// SIMATIC S7-200 project (STEP 7-Micro/WIN), CPU 224XP REL 02.01

SYMBOL_TABLE USER1
di_0_0           I0.0
di_0_1           I0.1
di_0_2           I0.2     // lazer_ON
di_0_3           I0.3
di_0_4           I0.4
di_0_5           I0.5
di_0_6           I0.6
di_0_7           I0.7
di_1_0           I1.0
di_1_1           I1.1
di_1_2           I1.2
di_1_3           I1.3
di_1_4           I1.4
di_1_5           I1.5
m0.0             M0.0
m0.1             M0.1
m0.2             M0.2
m0.3             M0.3
m0.4             M0.4
m0.5             M0.5
m0.6             M0.6
m0.7             M0.7
m1.0             M1.0
m1.1             M1.1
m1.2             M1.2
m1.3             M1.3
m1.4             M1.4
m1.5             M1.5
m1.6             M1.6
m1.7             M1.7
MB_DONE          M3.0
Port0_free_MB    M3.1
mb_start_delay   M3.2
reset_doze_nd1_all M4.0
reset_doze_nd2_all M4.1
reset_doze_all   M4.2
q_0_0            Q0.0
q_0_1            Q0.1
q_0_2            Q0.2
q_0_3            Q0.3
q_0_4            Q0.4
q_0_5            Q0.5
q_0_6            Q0.6
q_0_7            Q0.7
q_1_0            Q1.0
q_1_1            Q1.1
q_2_0            Q2.0
q_2_1            Q2.1
q_2_2            Q2.2
q_2_3            Q2.3
q_2_4            Q2.4
q_2_5            Q2.5
q_2_6            Q2.6
q_2_7            Q2.7
q_3_0            Q3.0
q_3_1            Q3.1
q_3_2            Q3.2
q_3_3            Q3.3
q_3_4            Q3.4
q_3_5            Q3.5
q_3_6            Q3.6
q_3_7            Q3.7
q_4_0            Q4.0
q_4_1            Q4.1
q_4_2            Q4.2
q_4_3            Q4.3
q_4_4            Q4.4
q_4_5            Q4.5
q_4_6            Q4.6
q_4_7            Q4.7
err_dh2          V50.3
err_LT1_min_dop  V50.4
err_LT1_max_dop  V50.5
err_memory       V50.6
err_one_param    V50.7
err_ai_FT1       V51.0
err_ai_FT2       V51.1
err_ai_LT1       V51.2
err_ai_PT1       V51.3
err_PT1_max_dop  V51.4
err_sa2_stop     V51.5
err_dh1_aft      V51.6
err_dh2_aft      V51.7
warn_LT1_min_work V54.0
warn_LT1_max_work V54.1
warn_PT1_min_work V54.2
warn_PT1_max_work V54.3
warn_reserv_nd1_start V54.4
warn_reserv_nd2_start V54.5
warn_port0_mb    V54.6
warn_port0_mb_init V54.7
MB_ERR_CODE_DONE VB12
err_one_param_item VB13
MB_ERR_CODE_INIT VB14
port0_mb_addr    VB15
port0_mb_parity  VB16
par27            VB300    // port0_mb_parity
par28            VB301    // port0_mb_addr
par29            VB302    // again_dh
par30            VB303
par31            VB304
par32            VB305
par33            VB306
I_16MA           VD66
port0_mb_baudrate VD154
par34            VD320    // port0_mb_baudrate
par35            VD324
par36            VD328
sum1             VD360
sum2             VD364
rez1             VD368
rez2             VD372
doze_nd1_from_start VD376
doze_nd1_all     VD380
doze_nd2_from_start VD384
doze_nd2_all     VD388
tmpp             VD392
ai_FT1           VW0
ai_FT2           VW2
ai_LT1           VW4
ai_PT1           VW6
g_errors_0       VW50
g_errors_1       VW52
g_warnings_0     VW54
g_warnings_1     VW56
MB_HR            VW58
I_3MA            VW60
I_4MA            VW62
mb_start_delay_value VW64
LT1_zero         VW70
LT1_range        VW72
LT1_min_work     VW74
LT1_max_work     VW76
LT1_min_dop      VW78
LT1_max_dop      VW80
PT1_zero         VW82
PT1_range        VW84
PT1_min_work     VW86
PT1_max_work     VW88
PT1_max_dop      VW90
FT1_range        VW92
FT2_range        VW94
time_out_dh      VW96
time_out_dh_s    VW98
reserve_nd_start_tout_s VW100
reserve_nd_start_tout VW102
mask_errors_0    VW106
mask_errors_1    VW108
mask_warnings_0  VW110
mask_warnings_1  VW112
nsh_timer_counter_sec VW114
nsh_work_time    VW116
nsh_cycle_time   VW118
again_dh         VW120
par01            VW200    // FT1_RANGE
par02            VW202    // FT2_RANGE
par03            VW204    // PT1_RANGE
par04            VW206    // LT1_RANGE
par05            VW208    // PT1_zero
par06            VW210    // LT1_zero
par07            VW212    // LT1_min_work
par08            VW214    // LT1_max_work
par09            VW216    // LT1_min_dop
par10            VW218    // LT1_max_dop
par11            VW220    // PT1_min_work
par12            VW222    // PT1_max_work
par13            VW224    // PT1_max_dop
par14            VW226    // nsh_work_time:VW66
par15            VW228    // nsh_cycle_time:VW68
par16            VW230    // reserve_nd_start_tout_s:VW100
par17            VW232    // time_out_dh_s:VW98
par18            VW234    // again_dh
par19            VW236
par20            VW238
par21            VW240
par22            VW242
par23            VW244
par24            VW246
par25            VW248
par26            VW250
flow             VW252
tmp              VW350
count            VW352
adder            VW354
total1           VW356
total2           VW358
END_SYMBOL_TABLE

SYMBOL_TABLE MB_HOLD
H_40001          VW500    // ai_FT1
H_40002          VW502    // ai_FT2
H_40003          VW504    // ai_LT1
H_40004          VW506    // ai_PT1
H_40005          VW508
H_40006          VW510
H_40007          VW512
H_40008          VW514
H_40009          VW516
H_40010          VW518
H_40011          VW520
H_40012          VW522
H_40013          VW524
H_40014          VW526
H_40015          VW528
H_40016          VW530
H_40017_0        V532.0   // лазер
H_40017_1        V532.1   // свет нло
H_40017_2        V532.2
H_40017_3        V532.3
H_40017_4        V532.4
H_40017_5        V532.5
H_40017_6        V532.6
H_40017_7        V532.7
H_40017_8        V533.0   // свет
H_40017_9        V533.1   // q0.1
H_40017_10       V533.2   // q0.2
H_40017_11       V533.3   // relay 16a
H_40017_12       V533.4   // q0.4
H_40017_13       V533.5   // светофор хранилище
H_40017_14       V533.6   // +12 под нло резерв
H_40017_15       V533.7   // дым п1
H_40018_0        V534.0   // red
H_40018_1        V534.1   // green
H_40018_2        V534.2   // blue
H_40018_3        V534.3   // вход в дезинфекцию
H_40018_4        V534.4   // жалюзи закрыть
H_40018_5        V534.5   // жалюзи открыть
H_40018_6        V534.6   // вход в квест
H_40018_7        V534.7   // уф лампы
H_40018_8        V535.0   // откр рубильник
H_40018_9        V535.1   // микроскоп
H_40018_10       V535.2   // нло движение
H_40018_11       V535.3   // помпа жизнеобесп
H_40018_12       V535.4   // red
H_40018_13       V535.5   // green
H_40018_14       V535.6   // blue
H_40018_15       V535.7   // вход в смотровую
H_40019_0        V536.0
H_40019_1        V536.1
H_40019_2        V536.2
H_40019_3        V536.3
H_40019_4        V536.4
H_40019_5        V536.5
H_40019_6        V536.6
H_40019_7        V536.7
H_40019_8        V537.0   // warn_LT1_min_work:V54.0
H_40019_9        V537.1   // warn_LT1_max_work:V54.1
H_40019_10       V537.2   // warn_PT1_min_work:V54.2
H_40019_11       V537.3   // warn_PT1_max_work:V54.3
H_40019_12       V537.4   // warn_reserv_nd1_start:V54.4
H_40019_13       V537.5   // warn_reserv_nd2_start:V54.5
H_40019_14       V537.6   // q_3_6:Q3.6 exit qvest
H_40019_15       V537.7   // warn_port0_mb_init:V54.7
H_40020_0        V538.0   // power_on:M1.0
H_40020_1        V538.1   // ND1:M1.1
H_40020_2        V538.2   // ND2:M1.2
H_40020_3        V538.3   // nsh_manual:M1.3
H_40020_4        V538.4   // nsh_mixer_mode:M1.7
H_40020_5        V538.5   // Both_nd_enable:M1.4
H_40020_6        V538.6   // nsh_mixer:M1.6
H_40020_7        V538.7   // nsh_current:M1.5
H_40020_8        V539.0   // modul 3 4.0
H_40020_9        V539.1   // modul 3 4.1
H_40020_10       V539.2   // modul 3.4.2
H_40020_11       V539.3   // modul 3.4.3
H_40020_12       V539.4   // modul 3.4.4
H_40020_13       V539.5   // modul 3.4.5
H_40020_14       V539.6   // modul 3.4.6
H_40020_15       V539.7   // modul 3.4.7
H_40021_0        V540.0
H_40021_1        V540.1
H_40022          VW542
H_40023_0        V544.0
H_40023_1        V544.1
H_40023_2        V544.2
H_40023_3        V544.3
H_40023_4        V544.4
H_40023_5        V544.5
H_40023_6        V544.6
H_40023_7        V544.7
H_40023_8        V545.0
H_40023_9        V545.1
H_40023_10       V545.2
H_40023_11       V545.3
H_40023_12       V545.4
H_40023_13       V545.5
H_40023_14       V545.6
H_40023_15       V545.7
H_40024_0        V546.0
H_40024_1        V546.1
H_40024_2        V546.2
H_40024_3        V546.3
H_40024_4        V546.4
H_40024_5        V546.5
H_40024_6        V546.6
H_40024_7        V546.7
H_40024_8        V547.0
H_40024_9        V547.1
H_40024_10       V547.2
H_40024_11       V547.3
H_40024_12       V547.4
H_40024_13       V547.5
H_40024_14       V547.6
H_40024_15       V547.7
Н_40025          VW548
Н_40026          VW550
Н_40027          VW552
H_40028          VW554
H_40029_0        V556.0
H_40029_1        V556.1
H_40029_2        V556.2
H_40029_3        V556.3
H_40029_4        V556.4
H_40029_5        V556.5
H_40029_6        V556.6
H_40029_7        V556.7
H_40029_8        V557.0
H_40029_9        V557.1
H_40029_10       V557.2
H_40029_11       V557.3
H_40029_12       V557.4
H_40029_13       V557.5
H_40029_14       V557.6
H_40029_15       V557.7
H_40030_0        V558.0   // --
H_40030_1        V558.1
H_40030_2        V558.2
H_40030_3        V558.3
H_40030_4        V558.4
H_40030_5        V558.5
H_40030_6        V558.6
H_40030_7        V558.7
H_40030_8        V559.0
H_40030_9        V559.1
H_40030_10       V559.2
H_40030_11       V559.3
H_40030_12       V559.4
H_40030_13       V559.5
H_40030_14       V559.6
H_40030_15       V559.7
END_SYMBOL_TABLE

SYMBOL_TABLE S7-200 Symbols
Always_On        SM0.0    // Always ON
First_Scan_On    SM0.1    // ON for the first scan cycle only
Clock_1s         SM0.5    // Clock pulse that is ON for 0.5 s, OFF for 0.5 s, for a duty cycle time of 1 s.
Pot0_Value       SMB28    // Set to value corresponding to analog adjustment 0.
END_SYMBOL_TABLE

ORGANIZATION_BLOCK MAIN:OB1
TITLE=PROGRAM COMMENTS
BEGIN
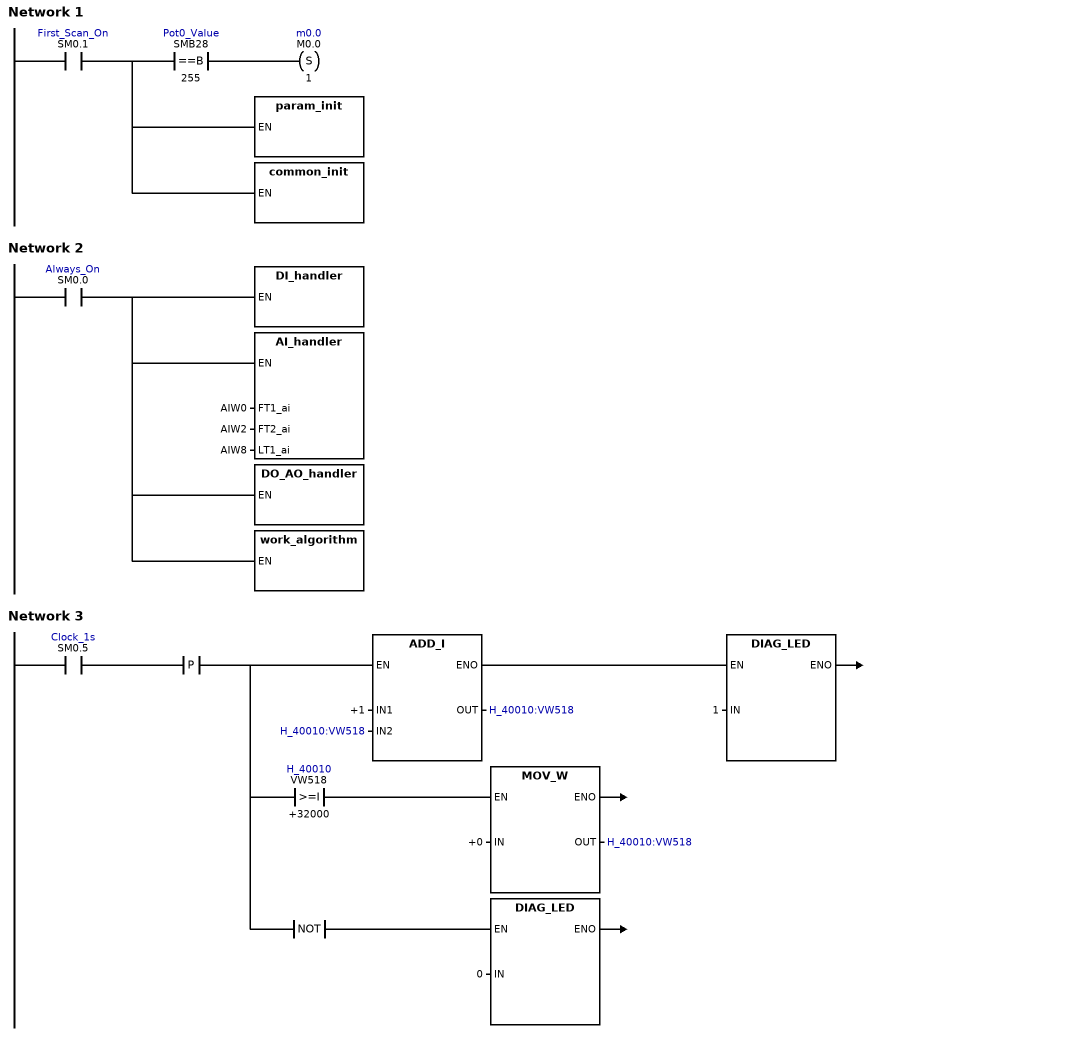
Network 1
LD     First_Scan_On:SM0.1
LPS
AB=    Pot0_Value:SMB28, 255
S      m0.0:M0.0, 1
LRD
CALL   param_init:SBR0
LPP
CALL   common_init:SBR1
Network 2
LD     Always_On:SM0.0
CALL   DI_handler:SBR2
CALL   AI_handler:SBR3, AIW0, AIW2, AIW8
CALL   DO_AO_handler:SBR6
CALL   work_algorithm:SBR4
Network 3
LD     Clock_1s:SM0.5
EU
LPS
+I     +1, H_40010:VW518
AENO
?32C   1
LRD
AW>=   H_40010:VW518, +32000
MOVW   +0, H_40010:VW518
LPP
NOT
?32C   0
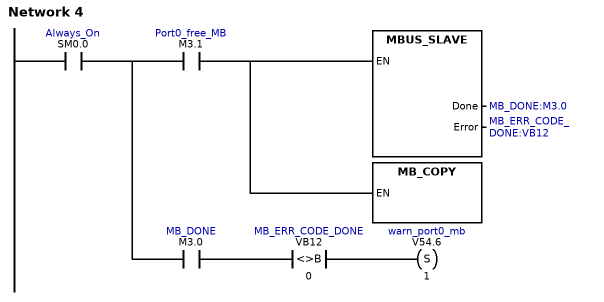
Network 4
LD     Always_On:SM0.0
LPS
A      Port0_free_MB:M3.1
CALL   MBUS_SLAVE:SBR13, MB_DONE:M3.0, MB_ERR_CODE_DONE:VB12
CALL   MB_COPY:SBR8
LPP
A      MB_DONE:M3.0
AB<>   MB_ERR_CODE_DONE:VB12, 0
S      warn_port0_mb:V54.6, 1
END_ORGANIZATION_BLOCK

SUBROUTINE_BLOCK param_init:SBR0
TITLE=
BEGIN
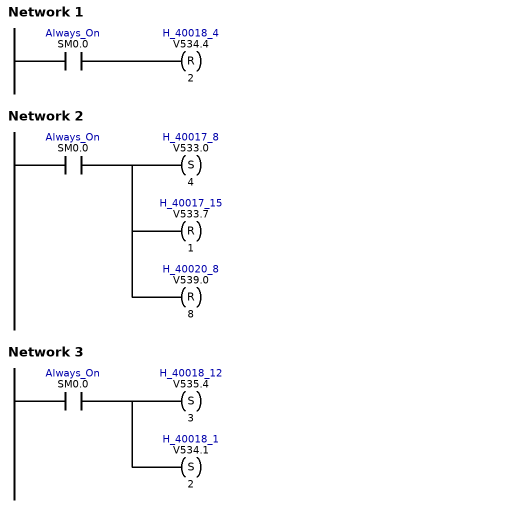
Network 1
LD     Always_On:SM0.0
R      H_40018_4:V534.4, 2
Network 2
LD     Always_On:SM0.0
S      H_40017_8:V533.0, 4
R      H_40017_15:V533.7, 1
R      H_40020_8:V539.0, 8
Network 3
LD     Always_On:SM0.0
S      H_40018_12:V535.4, 3
S      H_40018_1:V534.1, 2
END_SUBROUTINE_BLOCK

SUBROUTINE_BLOCK common_init:SBR1
TITLE=
BEGIN
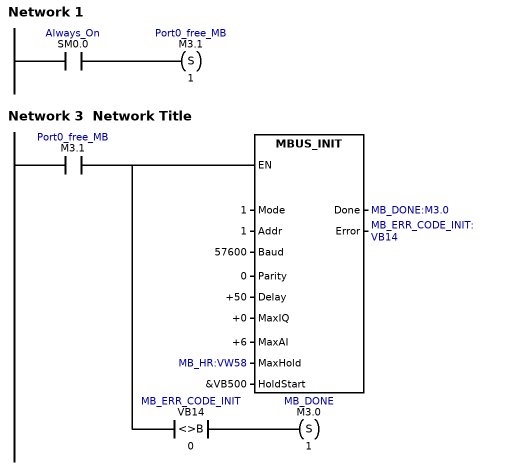
Network 1
LD     Always_On:SM0.0
S      Port0_free_MB:M3.1, 1
Network 3 // Network Title
LD     Port0_free_MB:M3.1
CALL   MBUS_INIT:SBR14, 1, 1, 57600, 0, +50, +0, +6, MB_HR:VW58, &VB500, MB_DONE:M3.0, MB_ERR_CODE_INIT:VB14
AB<>   MB_ERR_CODE_INIT:VB14, 0
S      MB_DONE:M3.0, 1
END_SUBROUTINE_BLOCK

SUBROUTINE_BLOCK AI_handler:SBR3
TITLE=SUBROUTINE COMMENTS
VAR_INPUT
FT1_ai:WORD;	// LW0 
FT2_ai:WORD;	// LW2 
LT1_ai:WORD;	// LW4 
END_VAR
BEGIN
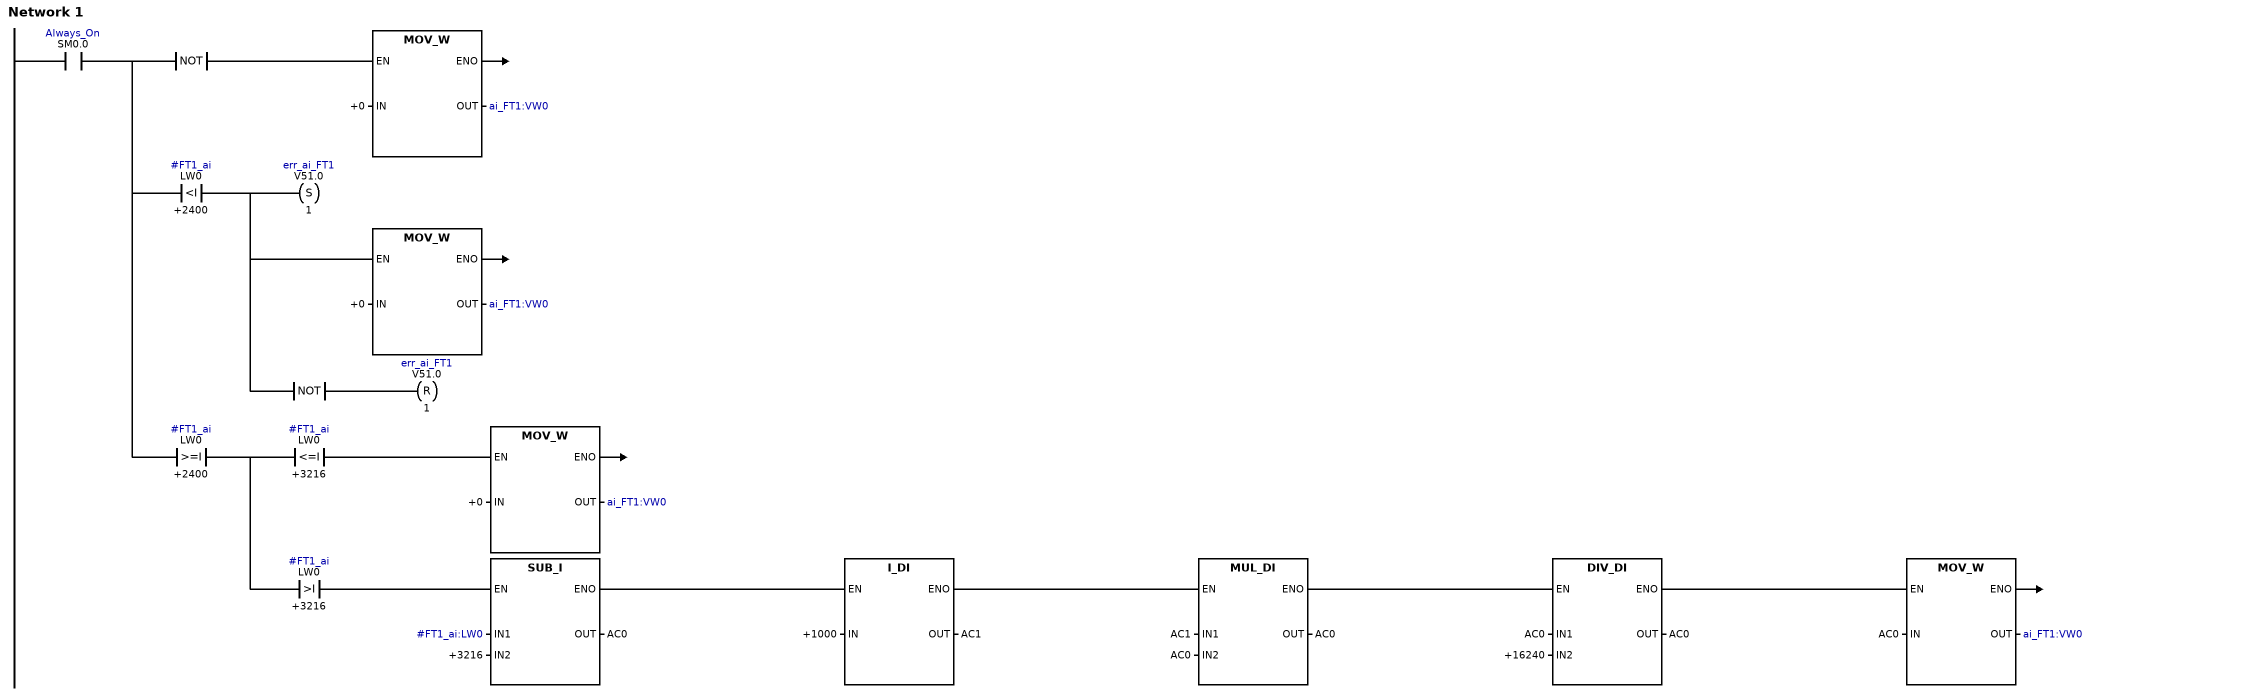
Network 1
LD     Always_On:SM0.0
LPS
NOT
MOVW   +0, ai_FT1:VW0
LRD
AW<    #FT1_ai:LW0, +2400
S      err_ai_FT1:V51.0, 1
MOVW   +0, ai_FT1:VW0
NOT
R      err_ai_FT1:V51.0, 1
LPP
AW>=   #FT1_ai:LW0, +2400
LPS
AW<=   #FT1_ai:LW0, +3216
MOVW   +0, ai_FT1:VW0
LPP
AW>    #FT1_ai:LW0, +3216
MOVW   #FT1_ai:LW0, AC0
AENO
-I     +3216, AC0
AENO
ITD    +1000, AC1
AENO
*D     AC1, AC0
AENO
/D     +16240, AC0
AENO
MOVW   AC0, ai_FT1:VW0
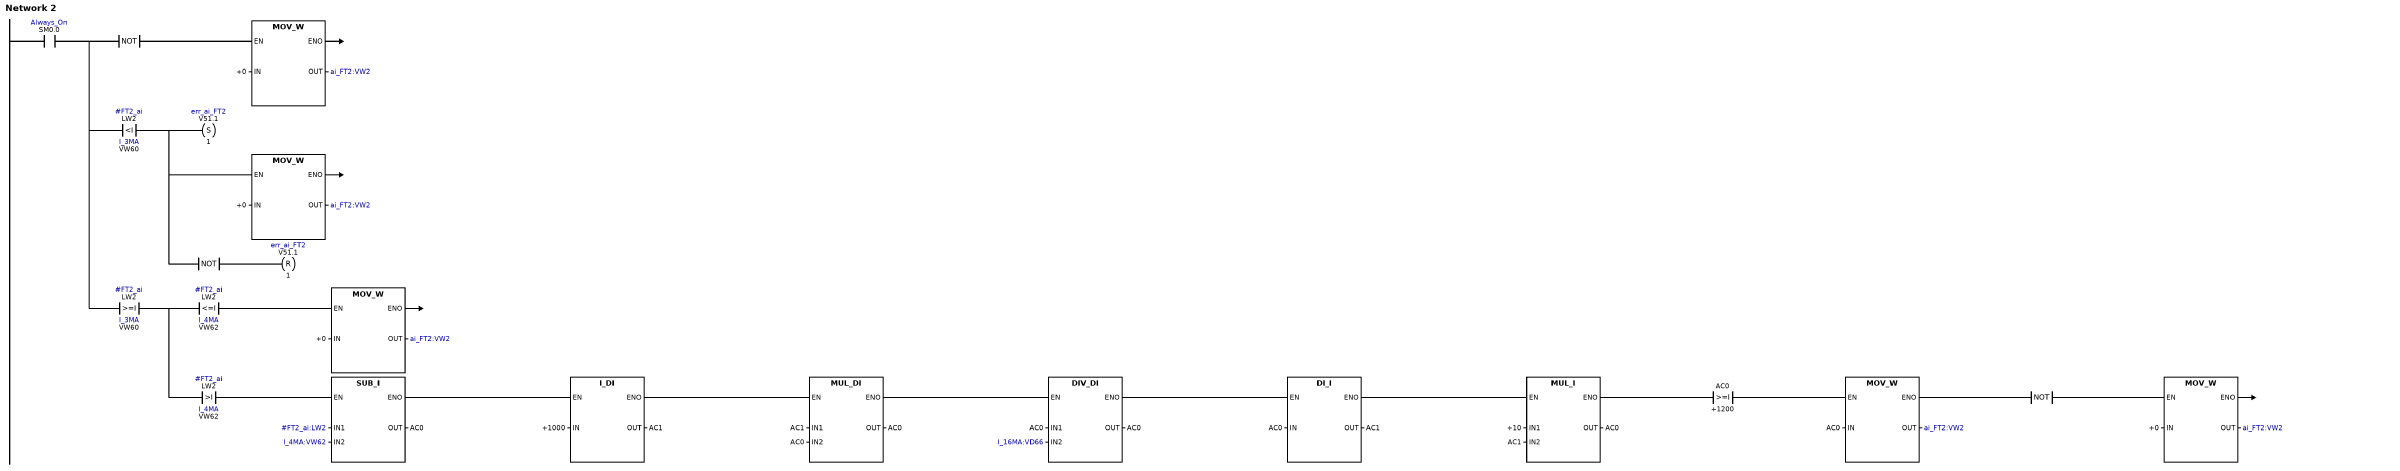
Network 2
LD     Always_On:SM0.0
LPS
NOT
MOVW   +0, ai_FT2:VW2
LRD
AW<    #FT2_ai:LW2, I_3MA:VW60
S      err_ai_FT2:V51.1, 1
MOVW   +0, ai_FT2:VW2
NOT
R      err_ai_FT2:V51.1, 1
LPP
AW>=   #FT2_ai:LW2, I_3MA:VW60
LPS
AW<=   #FT2_ai:LW2, I_4MA:VW62
MOVW   +0, ai_FT2:VW2
LPP
AW>    #FT2_ai:LW2, I_4MA:VW62
MOVW   #FT2_ai:LW2, AC0
AENO
-I     I_4MA:VW62, AC0
AENO
ITD    +1000, AC1
AENO
*D     AC1, AC0
AENO
/D     I_16MA:VD66, AC0
AENO
DTI    AC0, AC1
AENO
MOVW   +10, AC0
AENO
*I     AC1, AC0
AENO
AW>=   AC0, +1200
MOVW   AC0, ai_FT2:VW2
AENO
NOT
MOVW   +0, ai_FT2:VW2
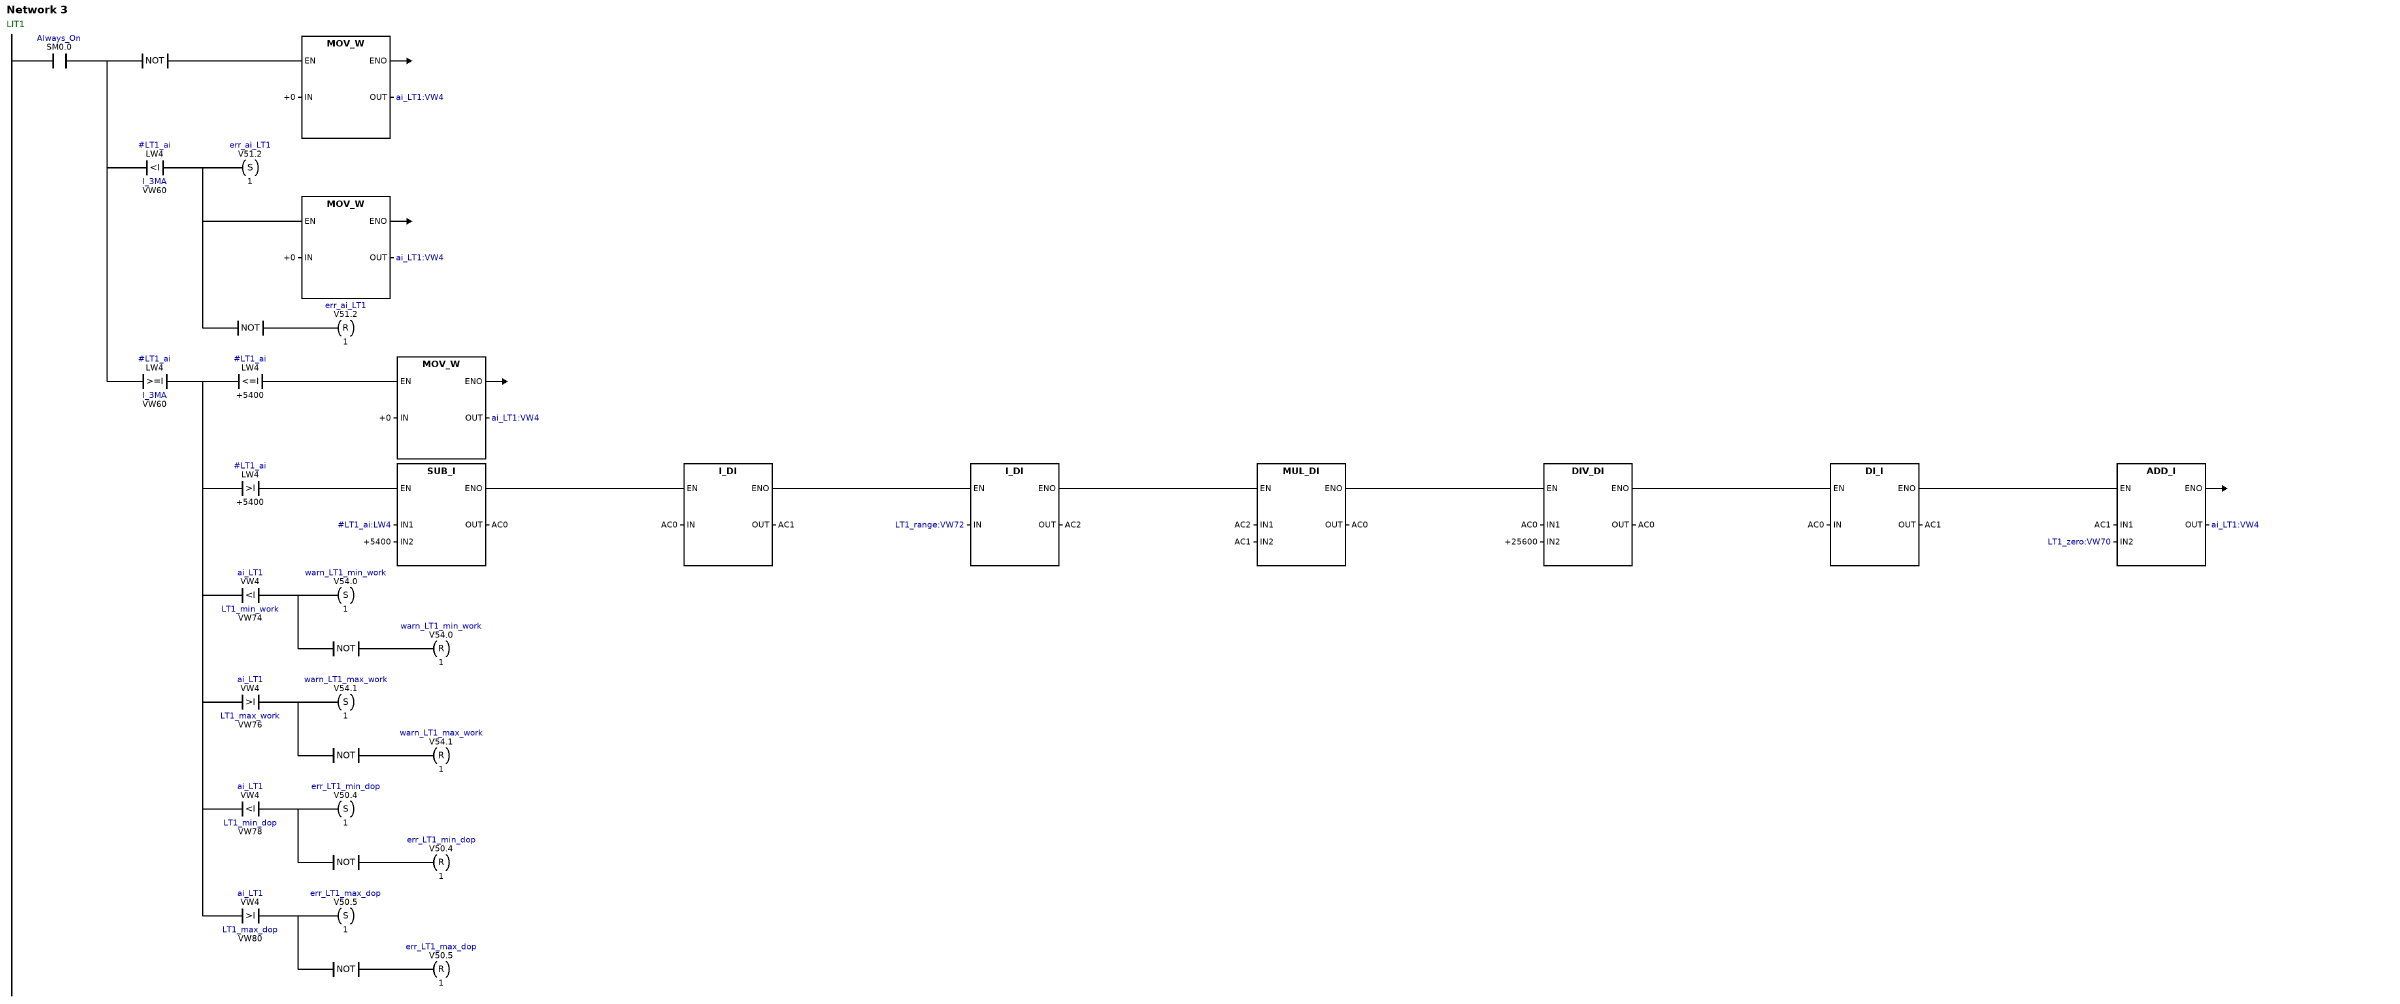
Network 3
//  LIT1
LD     Always_On:SM0.0
LPS
NOT
MOVW   +0, ai_LT1:VW4
LRD
AW<    #LT1_ai:LW4, I_3MA:VW60
S      err_ai_LT1:V51.2, 1
MOVW   +0, ai_LT1:VW4
NOT
R      err_ai_LT1:V51.2, 1
LPP
AW>=   #LT1_ai:LW4, I_3MA:VW60
LPS
AW<=   #LT1_ai:LW4, +5400
MOVW   +0, ai_LT1:VW4
LRD
AW>    #LT1_ai:LW4, +5400
MOVW   #LT1_ai:LW4, AC0
AENO
-I     +5400, AC0
AENO
ITD    AC0, AC1
AENO
ITD    LT1_range:VW72, AC2
AENO
MOVD   AC2, AC0
AENO
*D     AC1, AC0
AENO
/D     +25600, AC0
AENO
DTI    AC0, AC1
AENO
MOVW   AC1, ai_LT1:VW4
+I     LT1_zero:VW70, ai_LT1:VW4
LRD
AW<    ai_LT1:VW4, LT1_min_work:VW74
S      warn_LT1_min_work:V54.0, 1
NOT
R      warn_LT1_min_work:V54.0, 1
LRD
AW>    ai_LT1:VW4, LT1_max_work:VW76
S      warn_LT1_max_work:V54.1, 1
NOT
R      warn_LT1_max_work:V54.1, 1
LRD
AW<    ai_LT1:VW4, LT1_min_dop:VW78
S      err_LT1_min_dop:V50.4, 1
NOT
R      err_LT1_min_dop:V50.4, 1
LPP
AW>    ai_LT1:VW4, LT1_max_dop:VW80
S      err_LT1_max_dop:V50.5, 1
NOT
R      err_LT1_max_dop:V50.5, 1
END_SUBROUTINE_BLOCK

SUBROUTINE_BLOCK MB_COPY:SBR8
TITLE=КОММЕНТАРИИ ПОДПРОГРАММЫ
BEGIN
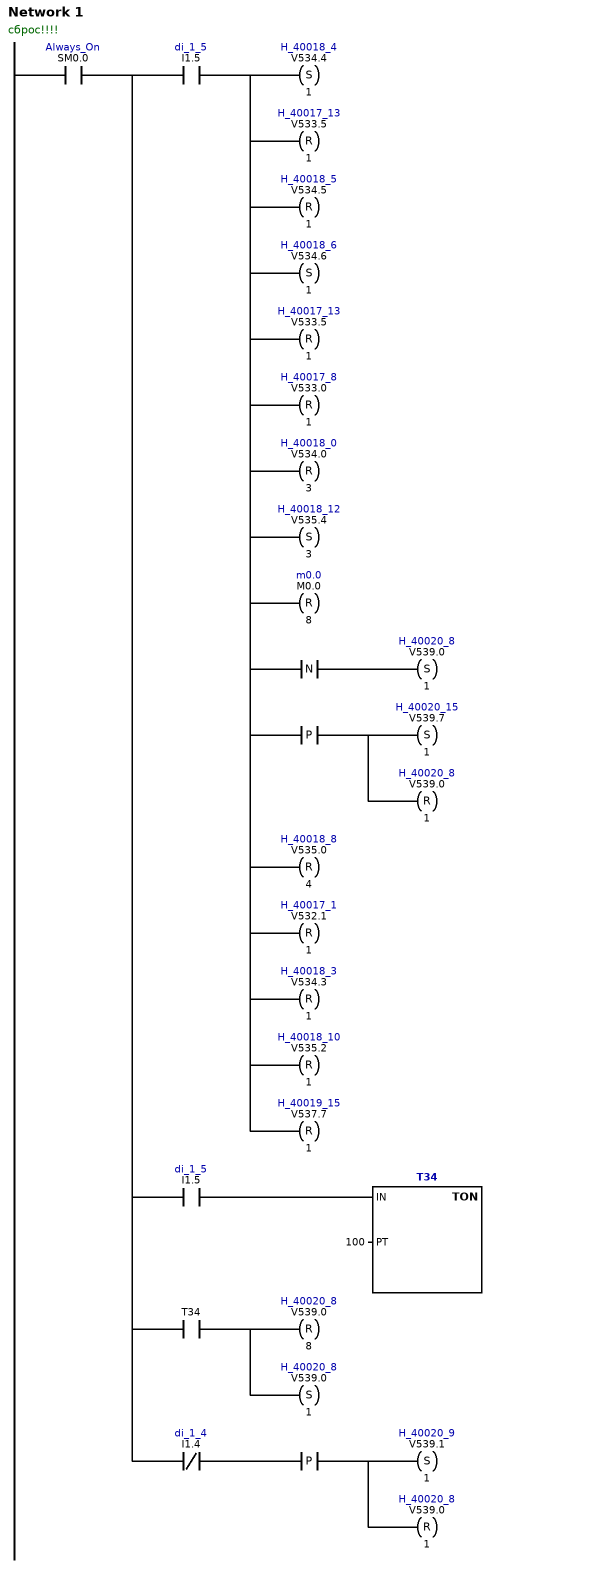
Network 1
// сброс!!!!
LD     Always_On:SM0.0
LPS
A      di_1_5:I1.5
LPS
S      H_40018_4:V534.4, 1
R      H_40017_13:V533.5, 1
R      H_40018_5:V534.5, 1
S      H_40018_6:V534.6, 1
R      H_40017_13:V533.5, 1
R      H_40017_8:V533.0, 1
R      H_40018_0:V534.0, 3
S      H_40018_12:V535.4, 3
R      m0.0:M0.0, 8
ED
S      H_40020_8:V539.0, 1
LRD
EU
S      H_40020_15:V539.7, 1
R      H_40020_8:V539.0, 1
LPP
R      H_40018_8:V535.0, 4
R      H_40017_1:V532.1, 1
R      H_40018_3:V534.3, 1
R      H_40018_10:V535.2, 1
R      H_40019_15:V537.7, 1
LPP
LPS
A      di_1_5:I1.5
TON    T34, 100
LRD
A      T34
R      H_40020_8:V539.0, 8
S      H_40020_8:V539.0, 1
LPP
AN     di_1_4:I1.4
EU
S      H_40020_9:V539.1, 1
R      H_40020_8:V539.0, 1
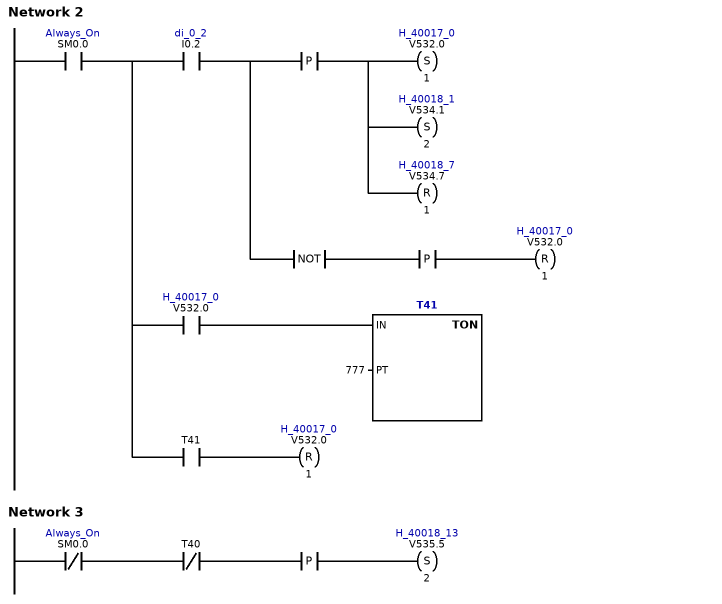
Network 2
LD     Always_On:SM0.0
LPS
A      di_0_2:I0.2
LPS
EU
S      H_40017_0:V532.0, 1
S      H_40018_1:V534.1, 2
R      H_40018_7:V534.7, 1
LPP
NOT
EU
R      H_40017_0:V532.0, 1
LPP
LPS
A      H_40017_0:V532.0
TON    T41, 777
LPP
A      T41
R      H_40017_0:V532.0, 1
Network 3
LDN    Always_On:SM0.0
AN     T40
EU
S      H_40018_13:V535.5, 2
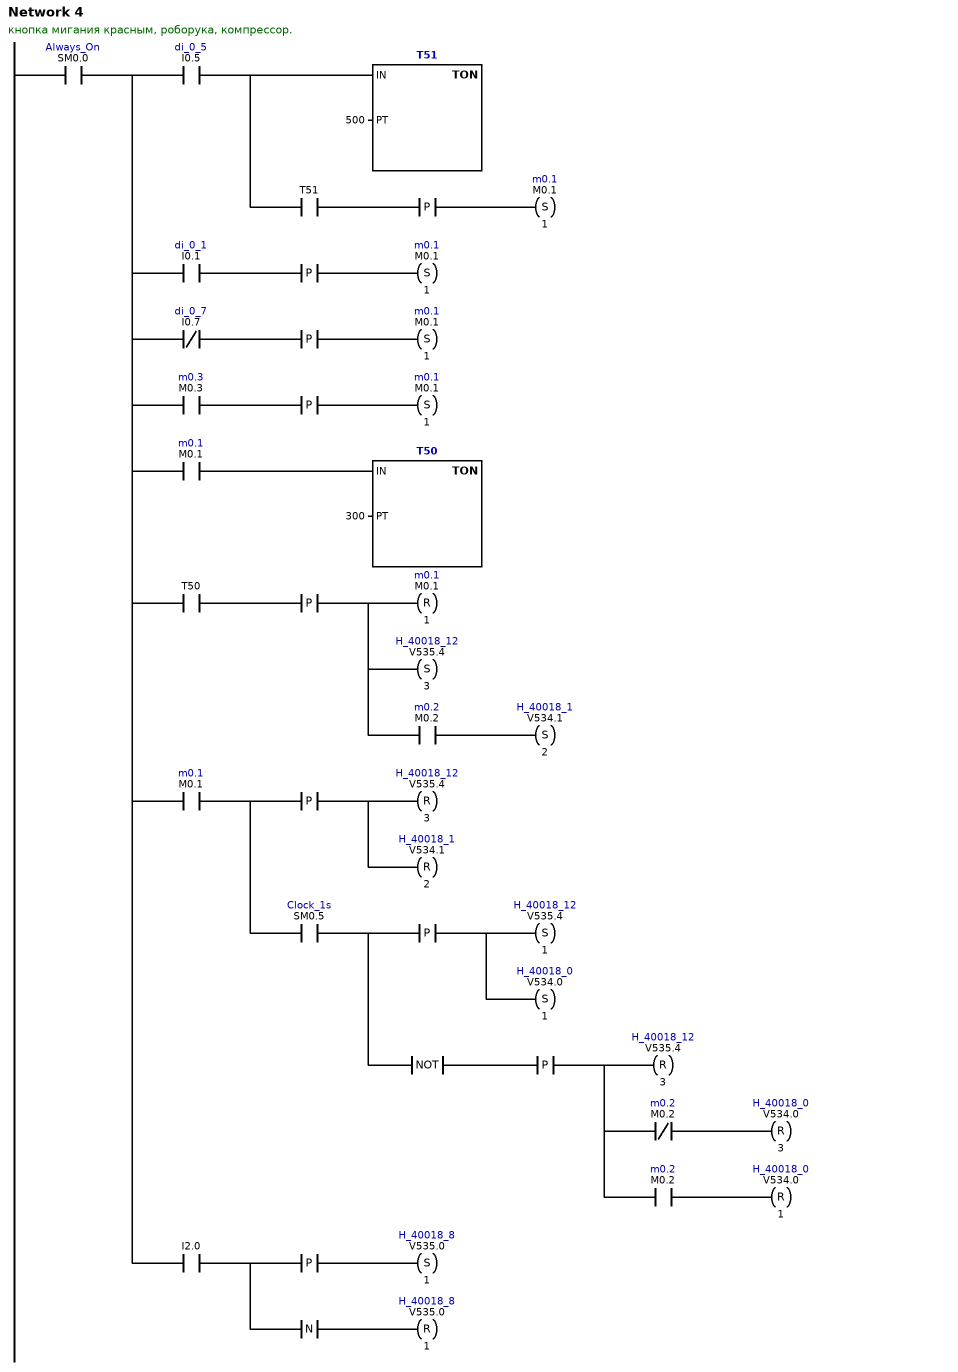
Network 4
// кнопка мигания красным, роборука, компрессор.
LD     Always_On:SM0.0
LPS
A      di_0_5:I0.5
TON    T51, 500
A      T51
EU
S      m0.1:M0.1, 1
LRD
LPS
A      di_0_1:I0.1
EU
S      m0.1:M0.1, 1
LRD
AN     di_0_7:I0.7
EU
S      m0.1:M0.1, 1
LRD
A      m0.3:M0.3
EU
S      m0.1:M0.1, 1
LPP
A      m0.1:M0.1
TON    T50, 300
LRD
A      T50
EU
R      m0.1:M0.1, 1
S      H_40018_12:V535.4, 3
A      m0.2:M0.2
S      H_40018_1:V534.1, 2
LRD
A      m0.1:M0.1
LPS
EU
R      H_40018_12:V535.4, 3
R      H_40018_1:V534.1, 2
LPP
A      Clock_1s:SM0.5
LPS
EU
S      H_40018_12:V535.4, 1
S      H_40018_0:V534.0, 1
LPP
NOT
EU
LPS
R      H_40018_12:V535.4, 3
AN     m0.2:M0.2
R      H_40018_0:V534.0, 3
LPP
A      m0.2:M0.2
R      H_40018_0:V534.0, 1
LPP
A      I2.0
LPS
EU
S      H_40018_8:V535.0, 1
LPP
ED
R      H_40018_8:V535.0, 1
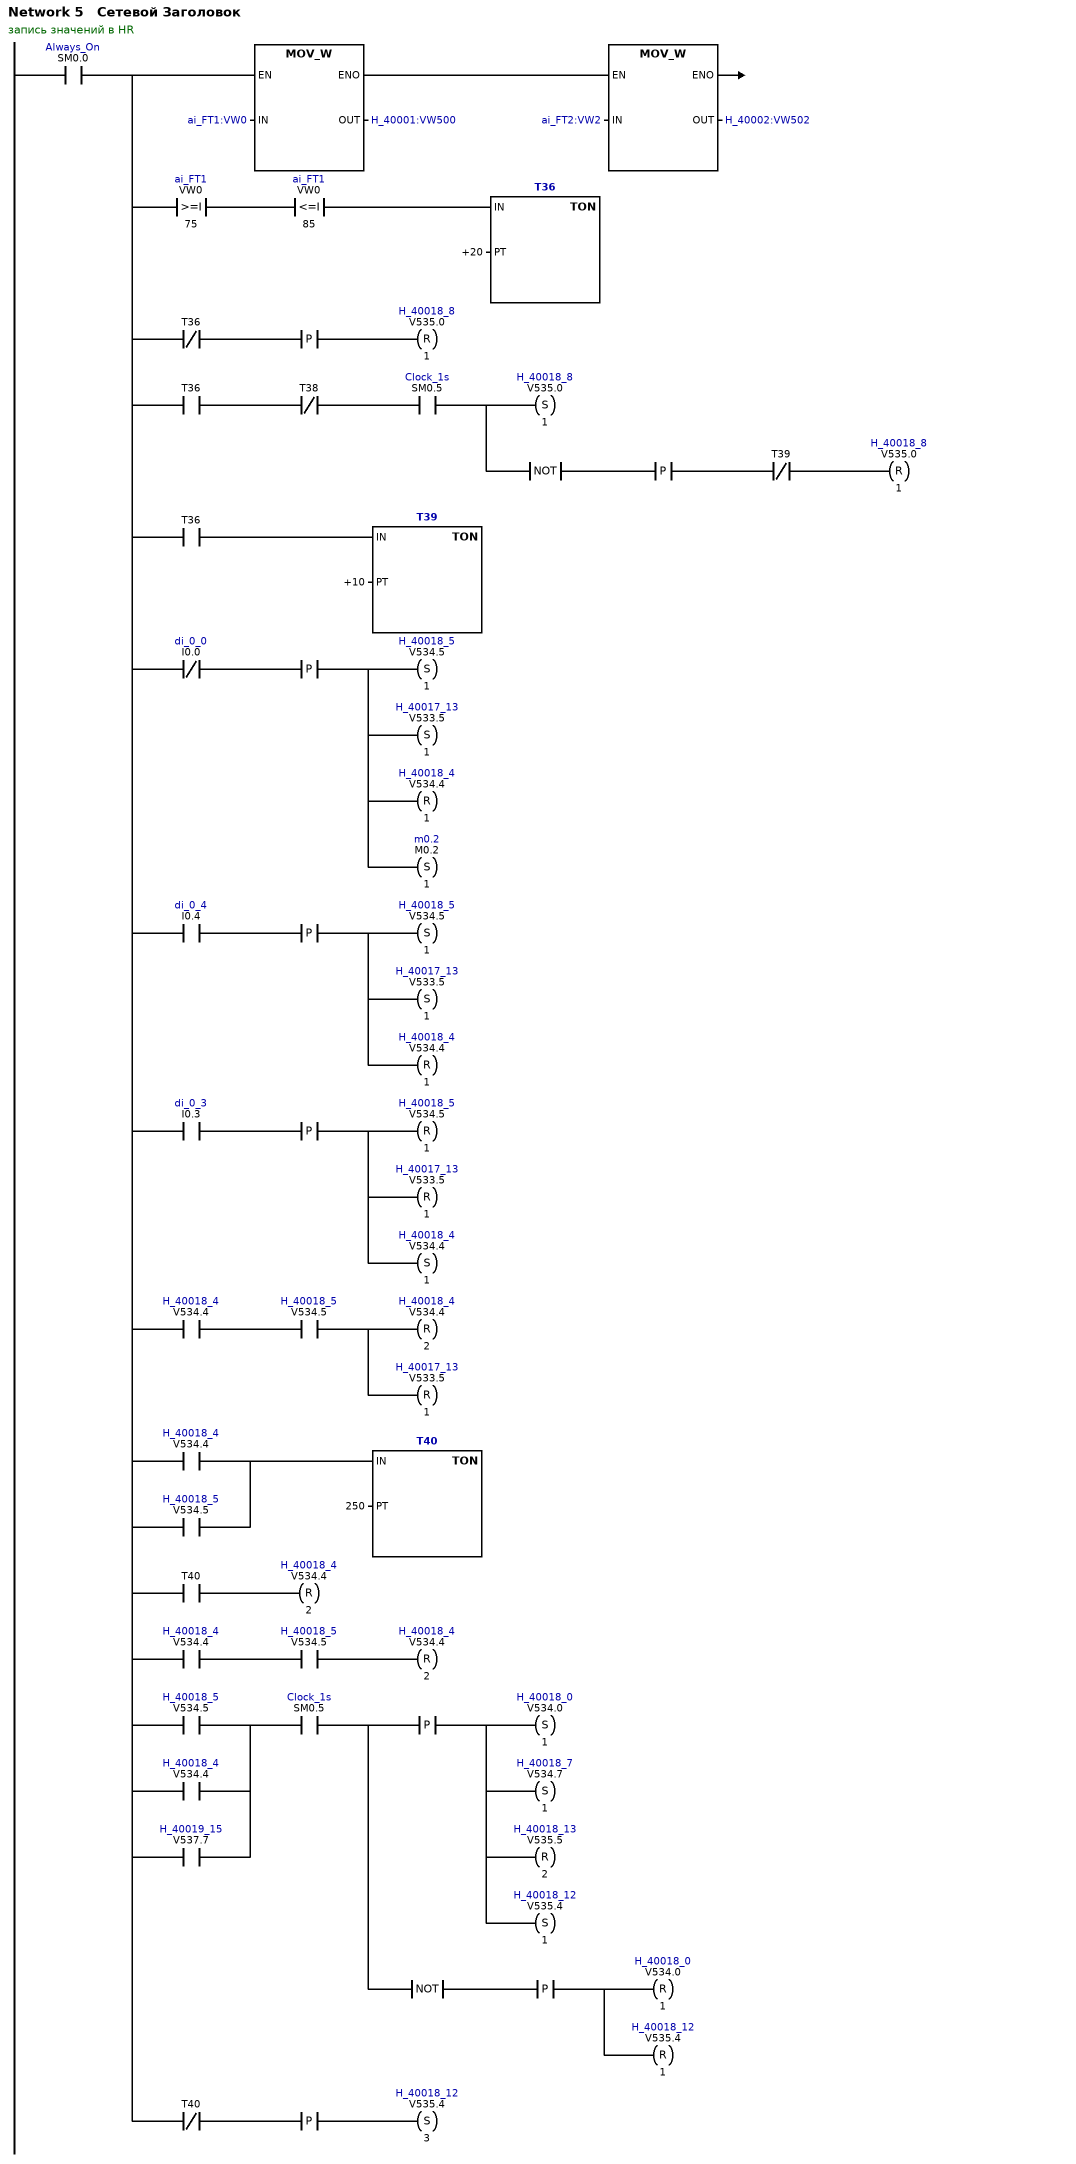
Network 5 //  Сетевой Заголовок
// запись значений в HR
LD     Always_On:SM0.0
LPS
MOVW   ai_FT1:VW0, H_40001:VW500
AENO
MOVW   ai_FT2:VW2, H_40002:VW502
LRD
AW>=   ai_FT1:VW0, 75
AW<=   ai_FT1:VW0, 85
TON    T36, +20
LRD
AN     T36
EU
R      H_40018_8:V535.0, 1
LRD
A      T36
AN     T38
A      Clock_1s:SM0.5
S      H_40018_8:V535.0, 1
NOT
EU
AN     T39
R      H_40018_8:V535.0, 1
LRD
A      T36
TON    T39, +10
LRD
AN     di_0_0:I0.0
EU
S      H_40018_5:V534.5, 1
S      H_40017_13:V533.5, 1
R      H_40018_4:V534.4, 1
S      m0.2:M0.2, 1
LRD
A      di_0_4:I0.4
EU
S      H_40018_5:V534.5, 1
S      H_40017_13:V533.5, 1
R      H_40018_4:V534.4, 1
LRD
A      di_0_3:I0.3
EU
R      H_40018_5:V534.5, 1
R      H_40017_13:V533.5, 1
S      H_40018_4:V534.4, 1
LRD
A      H_40018_4:V534.4
A      H_40018_5:V534.5
R      H_40018_4:V534.4, 2
R      H_40017_13:V533.5, 1
LRD
LD     H_40018_4:V534.4
O      H_40018_5:V534.5
ALD
TON    T40, 250
LRD
LPS
A      T40
R      H_40018_4:V534.4, 2
LPP
A      H_40018_4:V534.4
A      H_40018_5:V534.5
R      H_40018_4:V534.4, 2
LRD
LD     H_40018_5:V534.5
O      H_40018_4:V534.4
O      H_40019_15:V537.7
A      Clock_1s:SM0.5
ALD
LPS
EU
S      H_40018_0:V534.0, 1
S      H_40018_7:V534.7, 1
R      H_40018_13:V535.5, 2
S      H_40018_12:V535.4, 1
LPP
NOT
EU
R      H_40018_0:V534.0, 1
R      H_40018_12:V535.4, 1
LPP
AN     T40
EU
S      H_40018_12:V535.4, 3
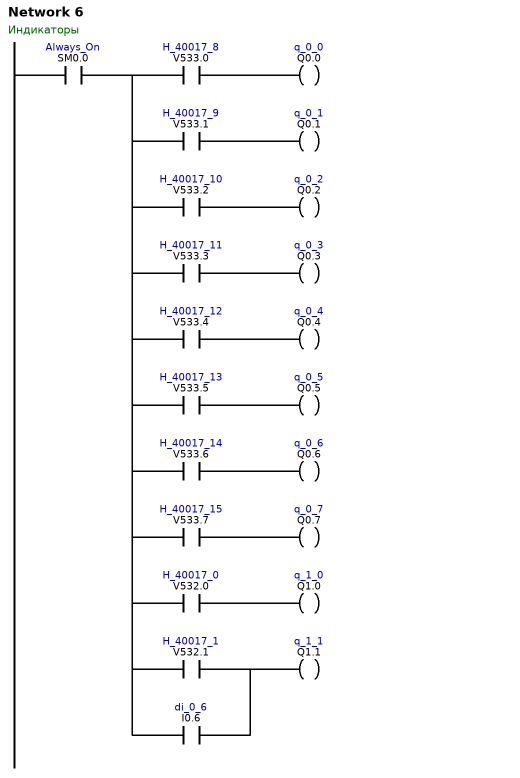
Network 6
//  Индикаторы
LD     Always_On:SM0.0
LPS
A      H_40017_8:V533.0
=      q_0_0:Q0.0
LRD
A      H_40017_9:V533.1
=      q_0_1:Q0.1
LRD
A      H_40017_10:V533.2
=      q_0_2:Q0.2
LRD
A      H_40017_11:V533.3
=      q_0_3:Q0.3
LRD
A      H_40017_12:V533.4
=      q_0_4:Q0.4
LRD
A      H_40017_13:V533.5
=      q_0_5:Q0.5
LRD
A      H_40017_14:V533.6
=      q_0_6:Q0.6
LRD
A      H_40017_15:V533.7
=      q_0_7:Q0.7
LRD
A      H_40017_0:V532.0
=      q_1_0:Q1.0
LPP
LD     H_40017_1:V532.1
O      di_0_6:I0.6
ALD
=      q_1_1:Q1.1
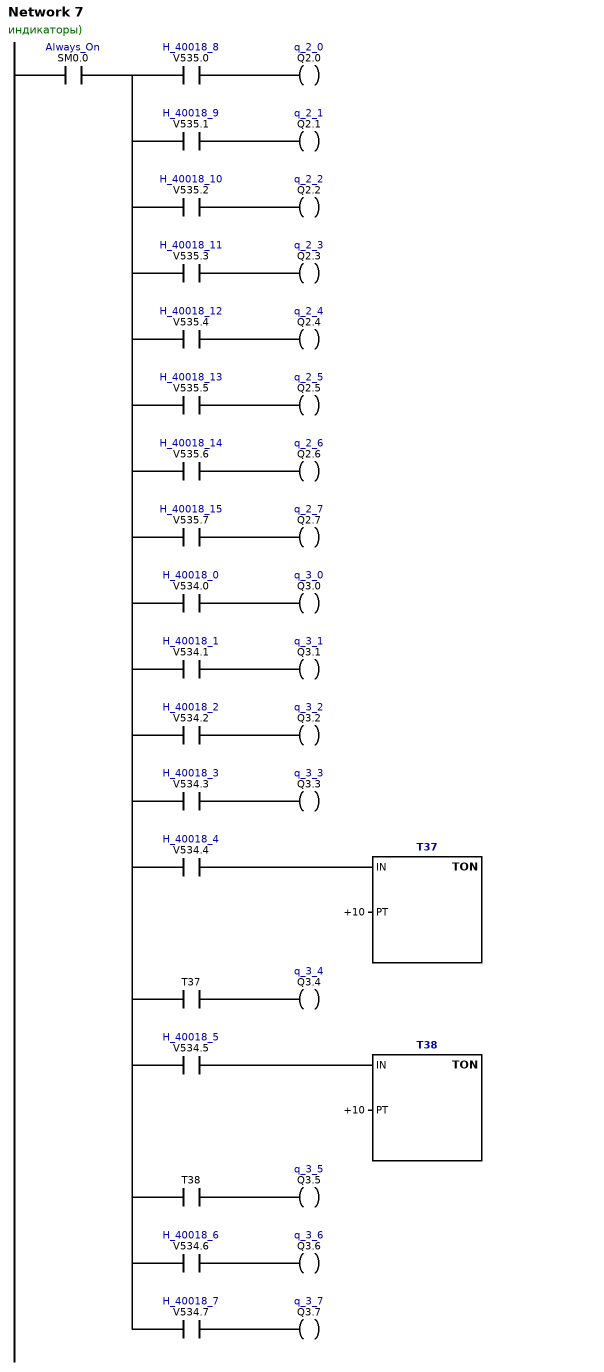
Network 7
//  индикаторы)
LD     Always_On:SM0.0
LPS
A      H_40018_8:V535.0
=      q_2_0:Q2.0
LRD
A      H_40018_9:V535.1
=      q_2_1:Q2.1
LRD
A      H_40018_10:V535.2
=      q_2_2:Q2.2
LRD
A      H_40018_11:V535.3
=      q_2_3:Q2.3
LRD
A      H_40018_12:V535.4
=      q_2_4:Q2.4
LRD
A      H_40018_13:V535.5
=      q_2_5:Q2.5
LRD
A      H_40018_14:V535.6
=      q_2_6:Q2.6
LRD
A      H_40018_15:V535.7
=      q_2_7:Q2.7
LRD
A      H_40018_0:V534.0
=      q_3_0:Q3.0
LRD
A      H_40018_1:V534.1
=      q_3_1:Q3.1
LRD
A      H_40018_2:V534.2
=      q_3_2:Q3.2
LRD
A      H_40018_3:V534.3
=      q_3_3:Q3.3
LRD
A      H_40018_4:V534.4
TON    T37, +10
LRD
A      T37
=      q_3_4:Q3.4
LRD
A      H_40018_5:V534.5
TON    T38, +10
LRD
A      T38
=      q_3_5:Q3.5
LRD
A      H_40018_6:V534.6
=      q_3_6:Q3.6
LPP
A      H_40018_7:V534.7
=      q_3_7:Q3.7
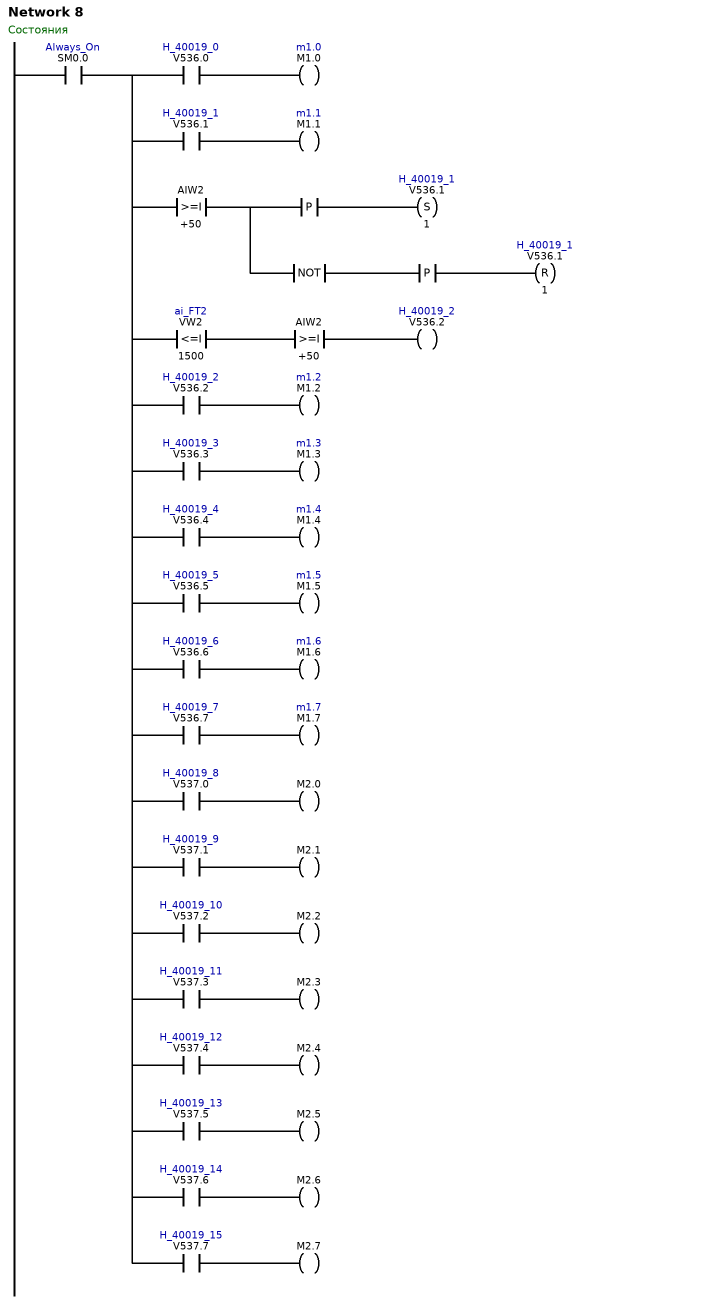
Network 8
//  Состояния
LD     Always_On:SM0.0
LPS
A      H_40019_0:V536.0
=      m1.0:M1.0
LRD
A      H_40019_1:V536.1
=      m1.1:M1.1
LRD
AW>=   AIW2, +50
LPS
EU
S      H_40019_1:V536.1, 1
LPP
NOT
EU
R      H_40019_1:V536.1, 1
LPP
LPS
AW<=   ai_FT2:VW2, 1500
AW>=   AIW2, +50
=      H_40019_2:V536.2
LRD
A      H_40019_2:V536.2
=      m1.2:M1.2
LRD
A      H_40019_3:V536.3
=      m1.3:M1.3
LRD
A      H_40019_4:V536.4
=      m1.4:M1.4
LRD
A      H_40019_5:V536.5
=      m1.5:M1.5
LRD
A      H_40019_6:V536.6
=      m1.6:M1.6
LRD
A      H_40019_7:V536.7
=      m1.7:M1.7
LRD
A      H_40019_8:V537.0
=      M2.0
LRD
A      H_40019_9:V537.1
=      M2.1
LRD
A      H_40019_10:V537.2
=      M2.2
LRD
A      H_40019_11:V537.3
=      M2.3
LRD
A      H_40019_12:V537.4
=      M2.4
LRD
A      H_40019_13:V537.5
=      M2.5
LRD
A      H_40019_14:V537.6
=      M2.6
LPP
A      H_40019_15:V537.7
=      M2.7
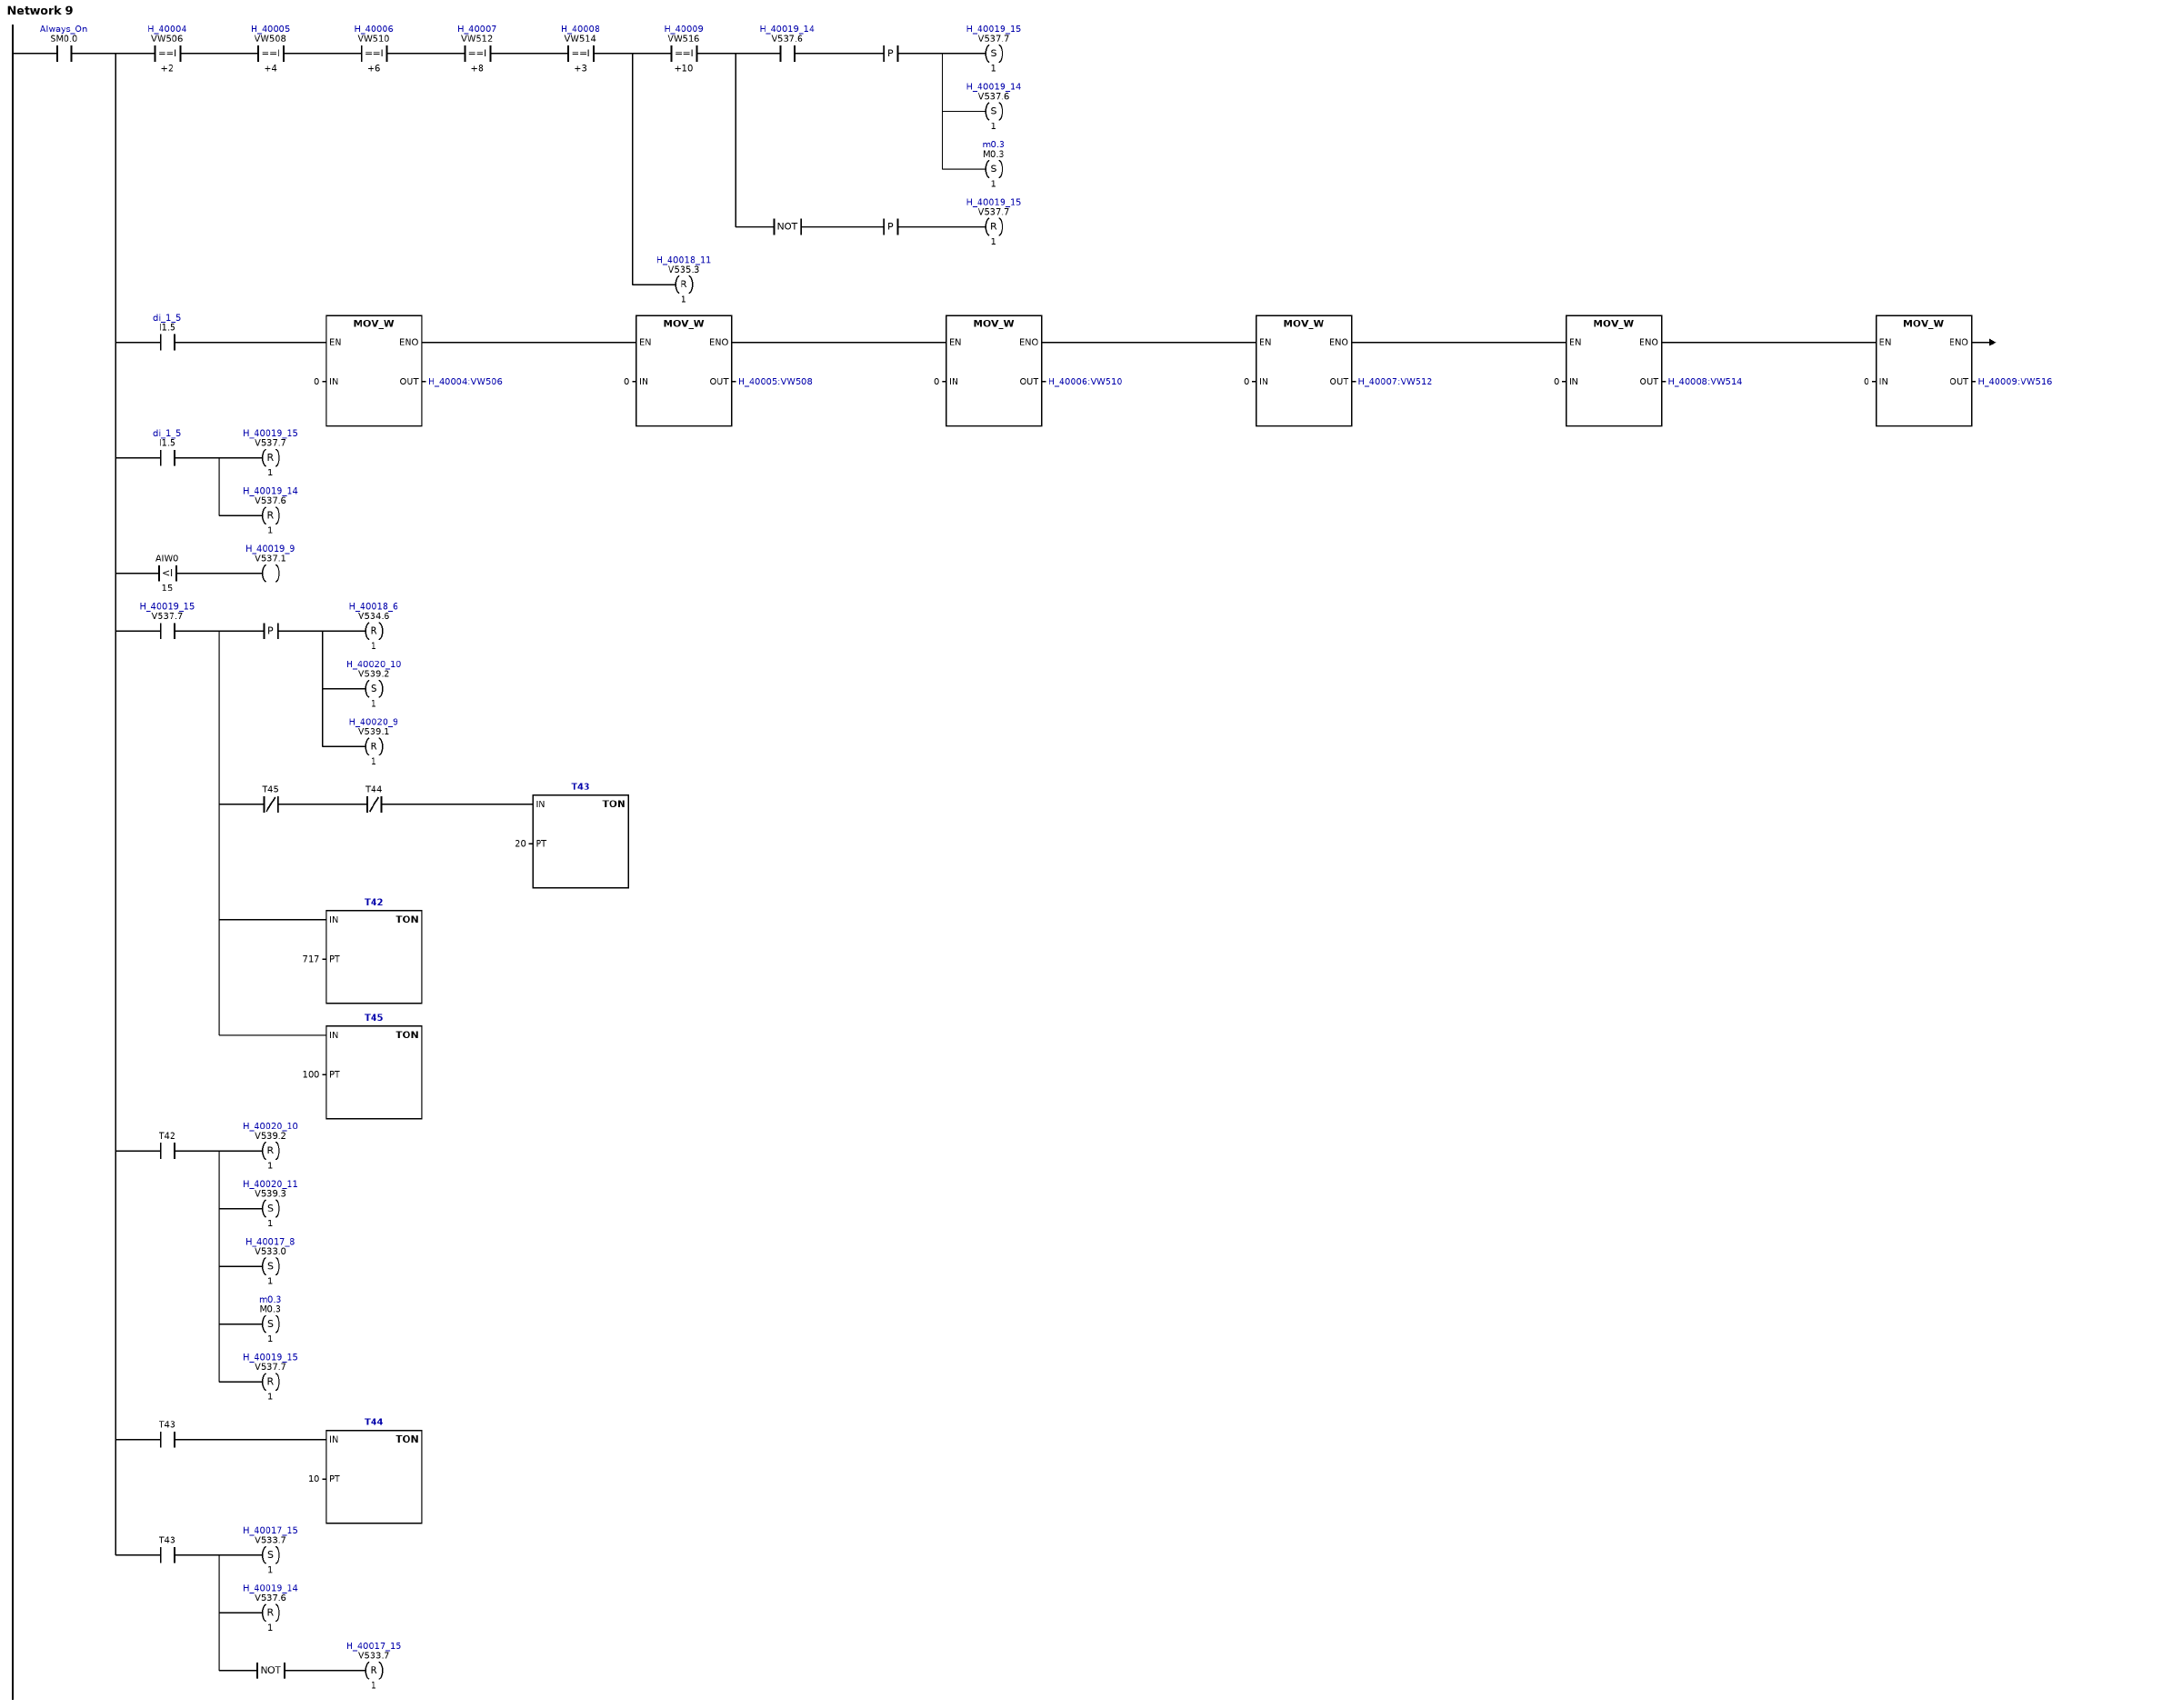
Network 9
LD     Always_On:SM0.0
LPS
AW=    H_40004:VW506, +2
AW=    H_40005:VW508, +4
AW=    H_40006:VW510, +6
AW=    H_40007:VW512, +8
AW=    H_40008:VW514, +3
LPS
AW=    H_40009:VW516, +10
LPS
A      H_40019_14:V537.6
EU
S      H_40019_15:V537.7, 1
S      H_40019_14:V537.6, 1
S      m0.3:M0.3, 1
LPP
NOT
EU
R      H_40019_15:V537.7, 1
LPP
R      H_40018_11:V535.3, 1
LPP
LPS
A      di_1_5:I1.5
MOVW   0, H_40004:VW506
AENO
MOVW   0, H_40005:VW508
AENO
MOVW   0, H_40006:VW510
AENO
MOVW   0, H_40007:VW512
AENO
MOVW   0, H_40008:VW514
AENO
MOVW   0, H_40009:VW516
LRD
A      di_1_5:I1.5
R      H_40019_15:V537.7, 1
R      H_40019_14:V537.6, 1
LRD
AW<    AIW0, 15
=      H_40019_9:V537.1
LRD
A      H_40019_15:V537.7
LPS
EU
R      H_40018_6:V534.6, 1
S      H_40020_10:V539.2, 1
R      H_40020_9:V539.1, 1
LPP
LPS
AN     T45
AN     T44
TON    T43, 20
LRD
TON    T42, 717
LPP
TON    T45, 100
LPP
LPS
A      T42
R      H_40020_10:V539.2, 1
S      H_40020_11:V539.3, 1
S      H_40017_8:V533.0, 1
S      m0.3:M0.3, 1
R      H_40019_15:V537.7, 1
LRD
A      T43
TON    T44, 10
LPP
A      T43
S      H_40017_15:V533.7, 1
R      H_40019_14:V537.6, 1
NOT
R      H_40017_15:V533.7, 1
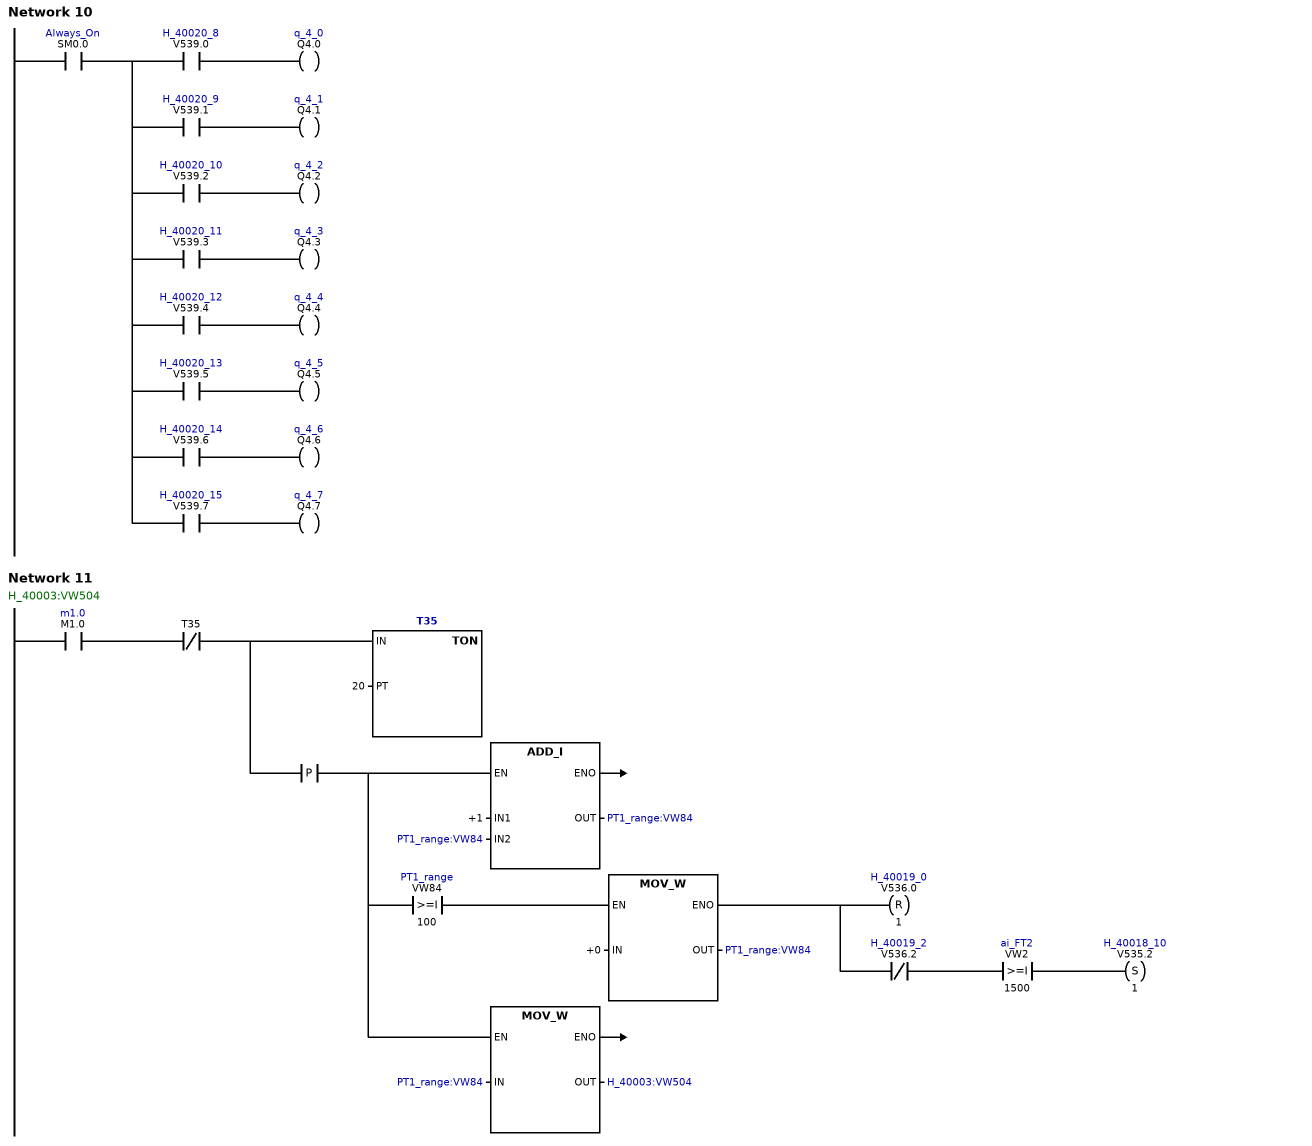
Network 10
LD     Always_On:SM0.0
LPS
A      H_40020_8:V539.0
=      q_4_0:Q4.0
LRD
A      H_40020_9:V539.1
=      q_4_1:Q4.1
LRD
A      H_40020_10:V539.2
=      q_4_2:Q4.2
LRD
A      H_40020_11:V539.3
=      q_4_3:Q4.3
LRD
A      H_40020_12:V539.4
=      q_4_4:Q4.4
LRD
A      H_40020_13:V539.5
=      q_4_5:Q4.5
LRD
A      H_40020_14:V539.6
=      q_4_6:Q4.6
LPP
A      H_40020_15:V539.7
=      q_4_7:Q4.7
Network 11
// H_40003:VW504
LD     m1.0:M1.0
AN     T35
TON    T35, 20
EU
LPS
+I     +1, PT1_range:VW84
AW>=   PT1_range:VW84, 100
MOVW   +0, PT1_range:VW84
AENO
R      H_40019_0:V536.0, 1
AN     H_40019_2:V536.2
AW>=   ai_FT2:VW2, 1500
S      H_40018_10:V535.2, 1
LPP
MOVW   PT1_range:VW84, H_40003:VW504
END_SUBROUTINE_BLOCK

// SBR12: protected block, not included

// SBR13: protected block, not included

// SBR14: protected block, not included

DATA_BLOCK_TAB USER1
BEGIN
//DATA PAGE COMMENTS
//Press F1 for help and example data page
         I_3MA, 16#12C0      //0960 для AI0,AI2
         I_4MA, 16#14FA      //0С80 для AI0,AI2  1900
         I_16MA, 16#8E94     //3200 для AI0,AI2 6400 было...(29000)7148
         MB_HR, 20           //100 bytes
         mb_start_delay_value, 30 //задержка вкл. МБ на 5 сек
END_DATA_BLOCK_TAB
